TYPE DOXControlChannel :
STRUCT
	{attribute addProperty Name "Control"}
	Control AT %Q* : stDOXcontrol;
END_STRUCT
END_TYPE

(* stored: Version 1.1.0.1, ProductVersion 3.1.4024.9
   DUT DOXControlChannel: Id {1e9bc842-a2a0-008a-1602-1378b52a2053} *)
